TYPE CamTableSelect_Status_typ EXTENDS MultiAxis_Status_typ :
	STRUCT
		
	END_STRUCT
END_TYPE

(* stored: Version 1.1.0.1, ProductVersion 3.1.4024.3
   DUT CamTableSelect_Status_typ: Id {f5fba353-4b0d-006b-129e-d32499623da9} *)
